PROGRAM MAIN
VAR
	myRobot:			TcA2B2Kitten;
	myRobotDigest:		TcA2B2KittenDigest;
	digestTest:			DigestTest;
//	cmdConnect:			BOOL;
//	connectCall:		PLCopenCall;
//	cmdGetRobotState: 	BOOL;
//	getRobotStateCall:	PLCopenCall;
END_VAR


// Call Robot Instance
//myRobot();
myRobotDigest();

UDPTest();

digestTest();

(*
/////////////////////////
// Connect

IF cmdConnect THEN
	myRobot.Connect(0, connectCall);
	cmdConnect := FALSE;
END_IF

connectCall();
connectCall.Execute := 0;

// Process command result
IF connectCall.Done THEN
	LogMessage(0, 'Connection Established');
ELSIF connectCall.Error THEN 
	LogMessage(0, 'Connection command error');
ELSIF connectCall.CommandAborted THEN 
	LogMessage(0, 'Connection command aborted');
END_IF

/////////////////////////
// Get Robot State

IF cmdGetRobotState THEN
	myRobot.GetRobotState(getRobotStateCall);
	cmdGetRobotState := FALSE;
END_IF

getRobotStateCall();
getRobotStateCall.Execute := 0;

// Process command result
IF getRobotStateCall.Done THEN
	LogMessage(0, 'GetRobotState Done');
ELSIF getRobotStateCall.Error THEN 
	LogMessage(0, 'GetRobotState command error');
ELSIF getRobotStateCall.CommandAborted THEN 
	LogMessage(0, 'GetRobotState command aborted');
END_IF
*)

END_PROGRAM

(* stored: Version 1.1.0.1, ProductVersion 3.1.4024.12
   POU MAIN: Id {4538d9a0-54db-42fe-8559-12ac5bfe1677}, SpecialFunc None *)
